TYPE ST_ReceiveStatus :
STRUCT
	TransmitDone        :BOOL;   //数据发送完成
    ReceiveRequest      :BOOL;    
    InitAccepted        :BOOL;
    SndBufferFull       :BOOL;
    PutDataDone         :BOOL;
    InputLength         :USINT;
    TotalInputLength    :USINT;
	
END_STRUCT
END_TYPE

(* stored: Version 1.1.0.1, ProductVersion 3.1.4024.9
   DUT ST_ReceiveStatus: Id {c6f6727f-6a9d-4717-9185-bba370c636b4} *)
